{attribute 'GeneratedUsingTerminal: EK1122-0000-0018'}
{attribute addProperty BoxType "EK1122-0000-0018"}
{attribute addProperty Id "Beckhoff_EL29xxsub_EK1100EK1100_1FC0878B2"}
{attribute addProperty CRC "4055758829"}
{attribute addProperty Size "2"}
TYPE Beckhoff_EL29xxEK1122_F1BDF7ED EXTENDS EK1122_1FC0878B :
STRUCT
	{attribute addProperty Name "Beckhoff_EL29xxsub_EK1100"}
	{attribute addProperty PreviousPort "Beckhoff EL29xxEK1122 : D"}
	Beckhoff_EL29xxsub_EK1100 : EK1100_1FC0878B;
END_STRUCT
END_TYPE

(* stored: Version 1.2.0.0, ProductVersion 3.1.4024.9
   DUT Beckhoff_EL29xxEK1122_F1BDF7ED: Id {dc1ebeba-3e5b-4e71-a613-5956a7229335} *)
